// TIA Portal V19 export
TYPE "LAF_typePlasticRollerEm6ParametersInterface"
// stored: Access Published
   STRUCT
      configuration : "LAF_typeRollerEm1Parameters";
      commands : "LBC_typeInterfaceCommands";
      monitoring { S7_SetPoint := 'True'} : "LAF_typePlasticRollerEm6ProcessValues";
   END_STRUCT;
END_TYPE
